// Mitsubishi GX Works2 project: 생자 실린더 on off 동시동작   PLC: Q02/Q02H

PROGRAM MAIN
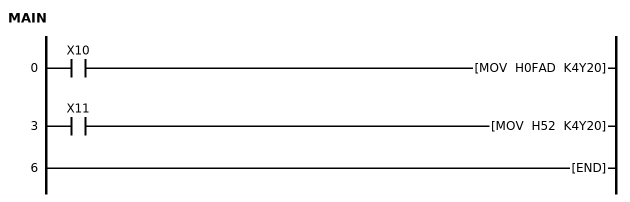
0     LD      X10
      MOV     H0FAD K4Y20
3     LD      X11
      MOV     H52 K4Y20
6     END
END_PROGRAM
